FUNCTION_BLOCK Q_ChildPosition (* Command change child position ( Part 6 - F.16 ) *)
  (* Standard: ISO 11783-6; Description: Copyright (c) 2022 HR Agrartechnik GmbH This program and the accompanying materials are made available under the terms of the Eclipse Public License 2.0 which is available at https://www.eclipse.org/legal/epl-2.0/ SPDX-License-Identifier: EPL-2.0 see Description Tab *)
  (* Version 1.0, 2022-07-08, Franz Höpfinger, HR Agrartechnik GmbH *)
  (* Documentation:
  Command change child position ( Part 6 - F.16 )
   The Change Child Location command is used to change the absolute position of an object.
   param[in] {objectID, uint16_t}
   Object ID
   param[in] {parentObjectID, uint16_t}
   Parent object ID
   param[in] {xPosition, uint16_t}
   New X position relative to the top left corner of parent object
   param[in] {yPosition, uint16_t}
   New Y position relative to the top left corner of parent object.
   Return Values: 
   int16_t
    - VT_E_NO_ERR (0) - OK
   - VT_E_OVERFLOW (-6) - buffer overflow
   - VT_E_NOACT (-8) - Command not possible in current state
   - VT_E_NO_INSTANCE (-21) - No VT client available
   - VT_E_ISO_INSTANCE_INVALID (-129) - Identifier for instance (connection) invalid
   - VT_E_NOT_ALIVE (-130) - Identifier for instance valid, but VT Dead.
  *)
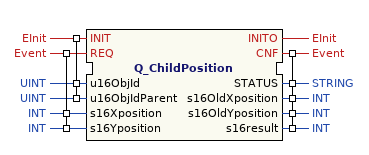
  EVENT_INPUT
    INIT : EInit WITH u16ObjId, u16ObjIdParent; (* Service Initialization *)
    REQ WITH s16Xposition, s16Yposition; (* Service Request *)
  END_EVENT
  EVENT_OUTPUT
    INITO : EInit; (* Initialization Confirm *)
    CNF WITH STATUS, s16OldYposition, s16OldXposition, s16result; (* Confirmation of Requested Service *)
  END_EVENT
  VAR_INPUT
    u16ObjId : UINT; (* Object ID *)
    u16ObjIdParent : UINT; (* Parent object ID *)
    s16Xposition : INT; (* New X position relative to the top left corner of parent object *)
    s16Yposition : INT; (* New Y position relative to the top left corner of parent object *)
  END_VAR
  VAR_OUTPUT
    STATUS : STRING; (* Service Status *)
    s16OldXposition : INT; (* Old X position relative to the top left corner of parent object *)
    s16OldYposition : INT; (* Old Y position relative to the top left corner of parent object *)
    s16result : INT; (* retval see description *)
  END_VAR
END_FUNCTION_BLOCK
